Fanuc KAREL source: source.kl

PROGRAM source
%NOLOCKGROUP

%INCLUDE source.klt

%INCLUDE source.klh

BEGIN
END source
